# EPICS substitutions: cg3-SE-PolyScience.substitutions
file PolyScience.db
{
pattern {S, TA, DN}
        {CG3, SE, PolyScience}
}

file ioc_sns.db
{
pattern {IOCNAME}
        {CG3:SE:PolyScience}
}
